// TIA Portal project "TiaPortal_TP_Final_V15.1" (V15.1)

(* hardware
DEVICE "S7-1200 station_1"  S7-1200 Station
   slot 0: "Rack_0"  S7-1200 Rack  Rack  V1.0
   slot 1: "PLC_1"  CPU 1214C AC/DC/Rly  6ES7 214-1BE30-0XB0  V2.0
   slot 3: "AQ 1x12BIT_1"  AQ1 signal board  6ES7 232-4HA30-0XB0  V1.0
*)

// ===== PLC "PLC_1"  CPU 1214C AC/DC/Rly =====

VAR_GLOBAL   // PLC tag table "Tabla de variables estándar"
   "Encendido" AT %M1.4 : Bool;
   "salida_duty_cycle" AT %QW80 : Int;
   "aceleracion_carrito" AT %MD58 : Real;
   "VEL1" AT %I0.2 : Bool;
   "VEL2" AT %I0.3 : Bool;
   "VEL3" AT %I0.4 : Bool;
   "VEL4" AT %I0.5 : Bool;
END_VAR

VAR_GLOBAL   // PLC tag table "Tabla de variables estándar_1"
   "System_Byte" AT %MB1 : Byte;
   "FirstScan" AT %M1.0 : Bool;
   "DiagStatusUpdate" AT %M1.1 : Bool;
   "AlwaysTRUE" AT %M1.2 : Bool;
   "AlwaysFALSE" AT %M1.3 : Bool;
   "Clock_Byte" AT %MB0 : Byte;
   "Clock_10Hz" AT %M0.0 : Bool;
   "Clock_5Hz" AT %M0.1 : Bool;
   "Clock_2.5Hz" AT %M0.2 : Bool;
   "Clock_2Hz" AT %M0.3 : Bool;
   "Clock_1.25Hz" AT %M0.4 : Bool;
   "Clock_1Hz" AT %M0.5 : Bool;
   "Clock_0.625Hz" AT %M0.6 : Bool;
   "Clock_0.5Hz" AT %M0.7 : Bool;
   "tcon_done_save" AT %M2.0 : Bool;
   "lectura_potenciometro" AT %IW66 : Word;
   "lectura_tacometro" AT %IW64 : Word;
   "PM" AT %I0.0 : Bool;
   "PP" AT %I0.1 : Bool;
   "lim_carreraA" AT %I1.3 : Bool;
   "lim_carreraB" AT %I1.2 : Bool;
   "posicion_carrito" AT %MD50 : Real;
   "velocidad_carrito" AT %MD54 : Real;
END_VAR

VAR_GLOBAL CONSTANT   // PLC tag table "Tabla de variables estándar_1"
   "Ninguno" : Pip := 65535;
   "Actualización automática" : Pip := 0;
   "IPP 1" : Pip := 1;
   "IPP 2" : Pip := 2;
   "IPP 3" : Pip := 3;
   "IPP 4" : Pip := 4;
   "IPP OB Servo" : Pip := 32768;
   "Local~MC" : Hw_SubModule := 51;
   "Local~Common" : Hw_SubModule := 50;
   "Local~Device" : Hw_Device := 32;
   "Local~Configuration" : Hw_SubModule := 33;
   "Local~Exec" : Hw_SubModule := 52;
   "Local(1)" : Hw_SubModule := 49;
   "Local~Interfaz_PROFINET_1(1)" : Hw_Interface := 64;
   "Local~Interfaz_PROFINET_1~Puerto_1(1)" : Hw_Interface := 65;
   "Local~Interfaz_PROFINET_1~Puerto_2" : Hw_Interface := 66;
   "Local~HSC_1(1)" : Hw_Hsc := 257;
   "Local~HSC_2(1)" : Hw_Hsc := 258;
   "Local~HSC_3(1)" : Hw_Hsc := 259;
   "Local~HSC_4(1)" : Hw_Hsc := 260;
   "Local~HSC_5(1)" : Hw_Hsc := 261;
   "Local~HSC_6(1)" : Hw_Hsc := 262;
   "Local~AI_2_AQ_2_1" : Hw_SubModule := 263;
   "Local~DI_14_DQ_10_1(1)" : Hw_SubModule := 264;
   "Local~Pulse_1(1)" : Hw_Pwm := 265;
   "Local~Pulse_2(1)" : Hw_Pwm := 266;
   "Local~Pulse_3" : Hw_Pwm := 267;
   "Local~Pulse_4" : Hw_Pwm := 268;
   "OB_Main(1)" : OB_PCYCLE := 1;
END_VAR

DATA_BLOCK "Datos_TSEND"   // DB2
{ S7_Optimized_Access := 'TRUE' }
VERSION : 0.1
   VAR
      data : Struct
         u : Real;
         aceleracion_carrito : Real;
         duty_cycle_pwm : Int;
      END_STRUCT;
   END_VAR
BEGIN
END_DATA_BLOCK

DATA_BLOCK "Comunicacion_DB"   // DB7
{ S7_Optimized_Access := 'TRUE' }
VERSION : 0.1
// stored: InstanceOfName Comunicacion
"Comunicacion"
BEGIN
END_DATA_BLOCK

DATA_BLOCK "Integrador_Velocidad_DB"   // DB9
{ S7_Optimized_Access := 'TRUE' }
VERSION : 0.1
// stored: InstanceOfName Integrador
"Integrador"
BEGIN
END_DATA_BLOCK

DATA_BLOCK "Controlador_DB"   // DB10
{ S7_Optimized_Access := 'TRUE' }
VERSION : 0.1
// stored: InstanceOfName Controlador
"Controlador"
BEGIN
END_DATA_BLOCK

DATA_BLOCK "Datos_General"   // DB11
{ S7_Optimized_Access := 'TRUE' }
VERSION : 0.1
   VAR
      MIN_ACEL_CARRITO : Real := -100.0;   // Aceleración mínima del carrito (porcentaje)
      MAX_ACEL_CARRITO : Real := 100.0;   // Aceleración máxima del carrito (porcentaje)
      MIN_VEL_CARRITO : Real := -100.0;   // Velocidad minima de motor (porcentaje)
      MAX_VEL_CARRITO : Real := 100.0;   // Velocidad maxima del carrito (porcentaje)
      MIN_POS_CARRITO : Real := -160.0;   // Posicion minima del carrito (en mm)
      MAX_POS_CARRITO : Real := 160.0;   // Posicion maxima del carrito (en mm)
      INIT_VEL_RESET : Real := 0.0;   // Velocidad inicial al resetear (porcentaje)
      INIT_POS_RESET : Real := 0.0;   // Posicion inicial al resetear (en mm)
      Tiempo_Muestreo : Real := 0.01;   // Tiempo en segundos del OB30
      LIM_INF_FILTRO_ACEL : Real := -5.0;   // Límite inferior del filtro para la aceleración
      LIM_SUP_FILTRO_ACEL : Real := 5.0;   // Límite superior del filtro para la aceleración
      SP_VEL_CARRITO : Real := 30.0;   // Set Point de velocidad del carrito
   END_VAR
BEGIN
END_DATA_BLOCK

DATA_BLOCK "Rutina_Identificacion_DB"   // DB12
{ S7_Optimized_Access := 'TRUE' }
VERSION : 0.1
// stored: InstanceOfName Rutina_Identificacion
"Rutina_Identificacion"
BEGIN
END_DATA_BLOCK

// folder: System blocks/Program resources

DATA_BLOCK "PLC_CONECTION_DB_"   // DB6
{ S7_Optimized_Access := 'TRUE' }
AUTHOR : SIMATIC
FAMILY : MC7Plus
NAME : TCON_Prm
VERSION : 1.0
// stored: InstanceOfName TCON_Param
"TCON_Param"
BEGIN
   ID := 2;
   REM_TSAP_ID[1] := B#16#07;
   REM_TSAP_ID[2] := B#16#D0;
   REM_STADDR[1] := 192;
   REM_STADDR[2] := 168;
   REM_STADDR[3] := 2;
   REM_STADDR[4] := 241;
END_DATA_BLOCK

// folder: (top level)

FUNCTION_BLOCK "Comunicacion"   // FB1, LAD
{ S7_Optimized_Access := 'TRUE' }
VERSION : 0.1
   VAR_INPUT
      acel_carrito : Real;
      vel_carrito : Real;
      salida_pwm : Int;
      vel_comandada : Real;
   END_VAR
   VAR CONSTANT
      LEN_DATA : UInt := 10;
   END_VAR
BEGIN

REGION Network 1
   // Se busca la conexión con la PC 1 vez por segundo
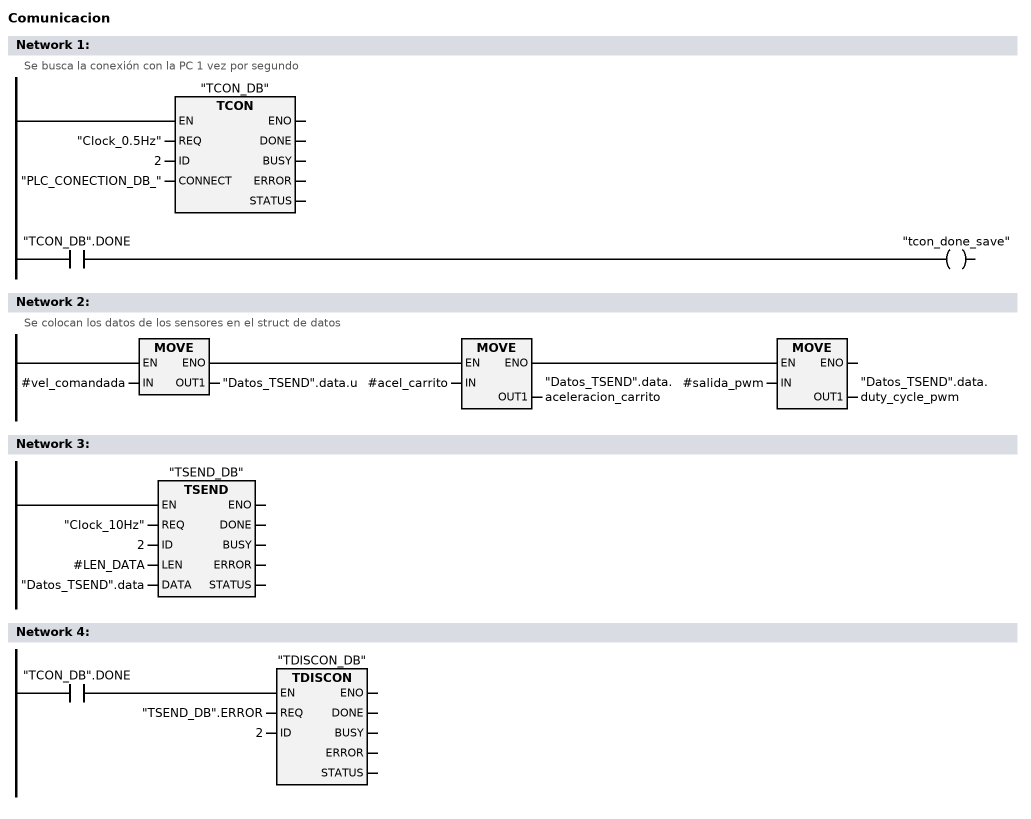
   "TCON_DB"(REQ := "Clock_0.5Hz", ID := 2, CONNECT := "PLC_CONECTION_DB_");   // TCON
   "tcon_done_save" := "TCON_DB".DONE;
END_REGION

REGION Network 2
   // Se colocan los datos de los sensores en el struct de datos
   RUNG wire#powerrail
      { S7_GenerateENO := "TRUE" } Move(in := #vel_comandada, out1 => "Datos_TSEND".data.u)
      { S7_GenerateENO := "TRUE" } Move(in := #acel_carrito, out1 => "Datos_TSEND".data.aceleracion_carrito)
      { S7_GenerateENO := "TRUE" } Move(in := #salida_pwm, out1 => "Datos_TSEND".data.duty_cycle_pwm)
   END_RUNG
   // the same network as SCL:
   // ENO of a box is taken as its EN; it also drops when the box reports an error
   "Datos_TSEND".data.u := #vel_comandada;
   "Datos_TSEND".data.aceleracion_carrito := #acel_carrito;
   "Datos_TSEND".data.duty_cycle_pwm := #salida_pwm;
END_REGION

REGION Network 3
   "TSEND_DB"(REQ := "Clock_10Hz", ID := 2, LEN := #LEN_DATA, DATA := "Datos_TSEND".data);   // TSEND
END_REGION

REGION Network 4
   IF "TCON_DB".DONE THEN
       "TDISCON_DB"(REQ := "TSEND_DB".ERROR, ID := 2);   // TDISCON
   END_IF;
END_REGION
END_FUNCTION_BLOCK

FUNCTION_BLOCK "Controlador"   // FB2, LAD
{ S7_Optimized_Access := 'TRUE' }
VERSION : 0.1
   VAR_INPUT
      SP_Velocidad : Real;   // en mm
      velocidad_actual_carrito : Real;   // porcentaje
      min_vel_perc_carrito : Real;   // porcentaje
      max_vel_perc_carrito : Real;   // porcentaje
   END_VAR
   VAR_OUTPUT
      salida_motor : Int;   // un valor entre n_cuenta_min y n_cuenta_max
   END_VAR
   VAR_TEMP
      vel_carrito_perc_pid : Real;
      vel : Real;
      vel_carrito_norm_pid : Real;
   END_VAR
   VAR CONSTANT
      n_cuenta_min : Int := 0;
      n_cuenta_max : Int := 27648;   // correspondiente a 16 bits del mapeo
   END_VAR
BEGIN

REGION Network 1
   // PID_VELOCIDAD
   // 
   // Input:
   // Recibe la velocidad actual del carrito en porcentaje y el setpoint en porcentaje (ambos son reales de -100.0 a 100.0)
   // 
   // Output:
   // Genera una salida porcentual entre -100.0%  y 100.0%, que es la velocidad a la cual debe accionarse el motor en reversa o en directa respectivamente.
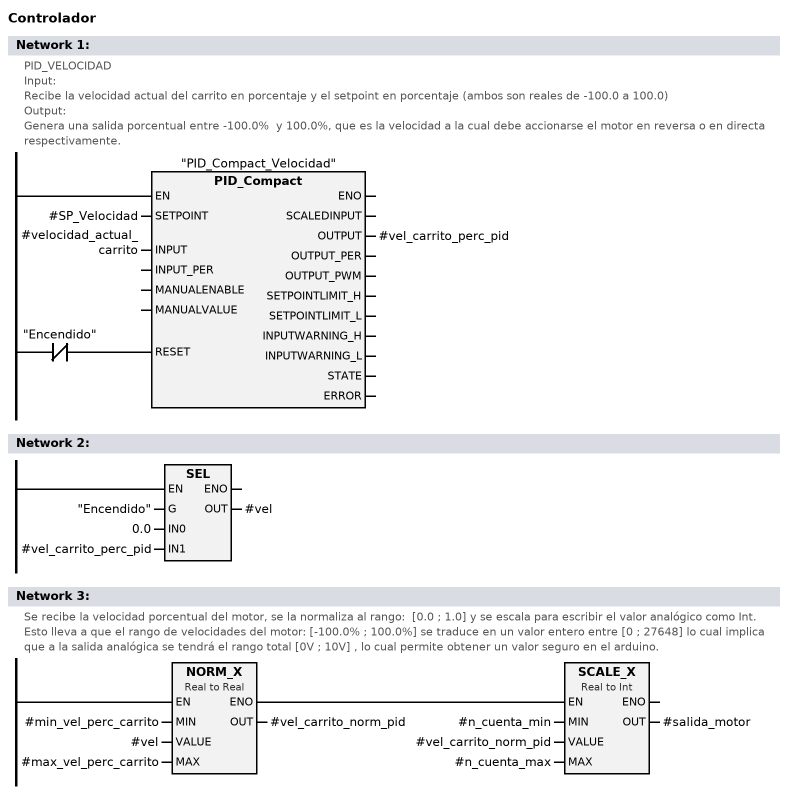
   "PID_Compact_Velocidad"(Setpoint := #SP_Velocidad,   // PID_Compact
                           Input := #velocidad_actual_carrito,
                           Reset := NOT "Encendido",
                           Output => #vel_carrito_perc_pid);
END_REGION

REGION Network 2
   #vel := SEL(G := "Encendido", IN0 := 0.0, IN1 := #vel_carrito_perc_pid);
END_REGION

REGION Network 3
   // Se recibe la velocidad porcentual del motor, se la normaliza al rango:  [0.0 ; 1.0] y se escala para escribir el valor analógico como Int.
   // Esto lleva a que el rango de velocidades del motor: [-100.0% ; 100.0%] se traduce en un valor entero entre [0 ; 27648] lo cual implica que a la salida analógica se tendrá el rango total [0V ; 10V] , lo cual permite obtener un valor seguro en el arduino.
   RUNG wire#powerrail
      { S7_Templates := "[SrcType := Real, DestType := Real]"; S7_GenerateENO := "TRUE" } Normalize(min := #min_vel_perc_carrito, value := #vel, max := #max_vel_perc_carrito, out => #vel_carrito_norm_pid)
      { S7_Templates := "[SrcType := Real, DestType := Int]"; S7_GenerateENO := "TRUE" } Scale(min := #n_cuenta_min, value := #vel_carrito_norm_pid, max := #n_cuenta_max, out => #salida_motor)
   END_RUNG
   // the same network as SCL:
   // ENO of a box is taken as its EN; it also drops when the box reports an error
   #vel_carrito_norm_pid := NORM_X(MIN := #min_vel_perc_carrito, VALUE := #vel, MAX := #max_vel_perc_carrito);
   #salida_motor := SCALE_X(MIN := #n_cuenta_min, VALUE := #vel_carrito_norm_pid, MAX := #n_cuenta_max);
END_REGION
END_FUNCTION_BLOCK

FUNCTION_BLOCK "Rutina_Identificacion"   // FB3, LAD
{ S7_Optimized_Access := 'TRUE' }
VERSION : 0.1
// Se fijó una tolerancia de 20mm para cada movimiento, además de un reinicio automático de la rutina
   VAR_INPUT
      posicion_carrito : Real;
      Encendido : Bool;
   END_VAR
   VAR_OUTPUT
      dc_pwm : Int := 13824;   // (detenido)
   END_VAR
   VAR
      Paso_1 : Bool;
      Paso_2 : Bool;
      Paso_3 : Bool;
      Paso_4 : Bool;
      Paso_5 : Bool;
      Paso_6 : Bool;
      Paso_7 : Bool;
      Paso_8 : Bool;
      Paso_9 : Bool;
      Paso_10 : Bool;
      Paso_11 : Bool;
      Paso_12 : Bool;
      Apagado : Bool;
      aux_encendido : Bool;
      IEC_Timer_Stop_Instance : TON_TIME;
      dc_stop : Int := 13824;   // (detenido)
      dc_f1 : Int := 20000;
      dc_f2 : Int := 19000;
      dc_f3 : Int := 18000;
      dc_b1 : Int := 6500;
      dc_b2 : Int := 7000;
      dc_b3 : Int := 7500;
      IEC_Timer_rutina : TON_TIME;
   END_VAR
   VAR_TEMP   // added for the SCL form of the ladder/FBD networks
      _w1 : Bool;
   END_VAR
   // IEC_Timer_Stop_Instance.PT := T#500ms;
   // IEC_Timer_rutina.PT := T#200ms;
BEGIN

REGION Network 1
   // Inicialización
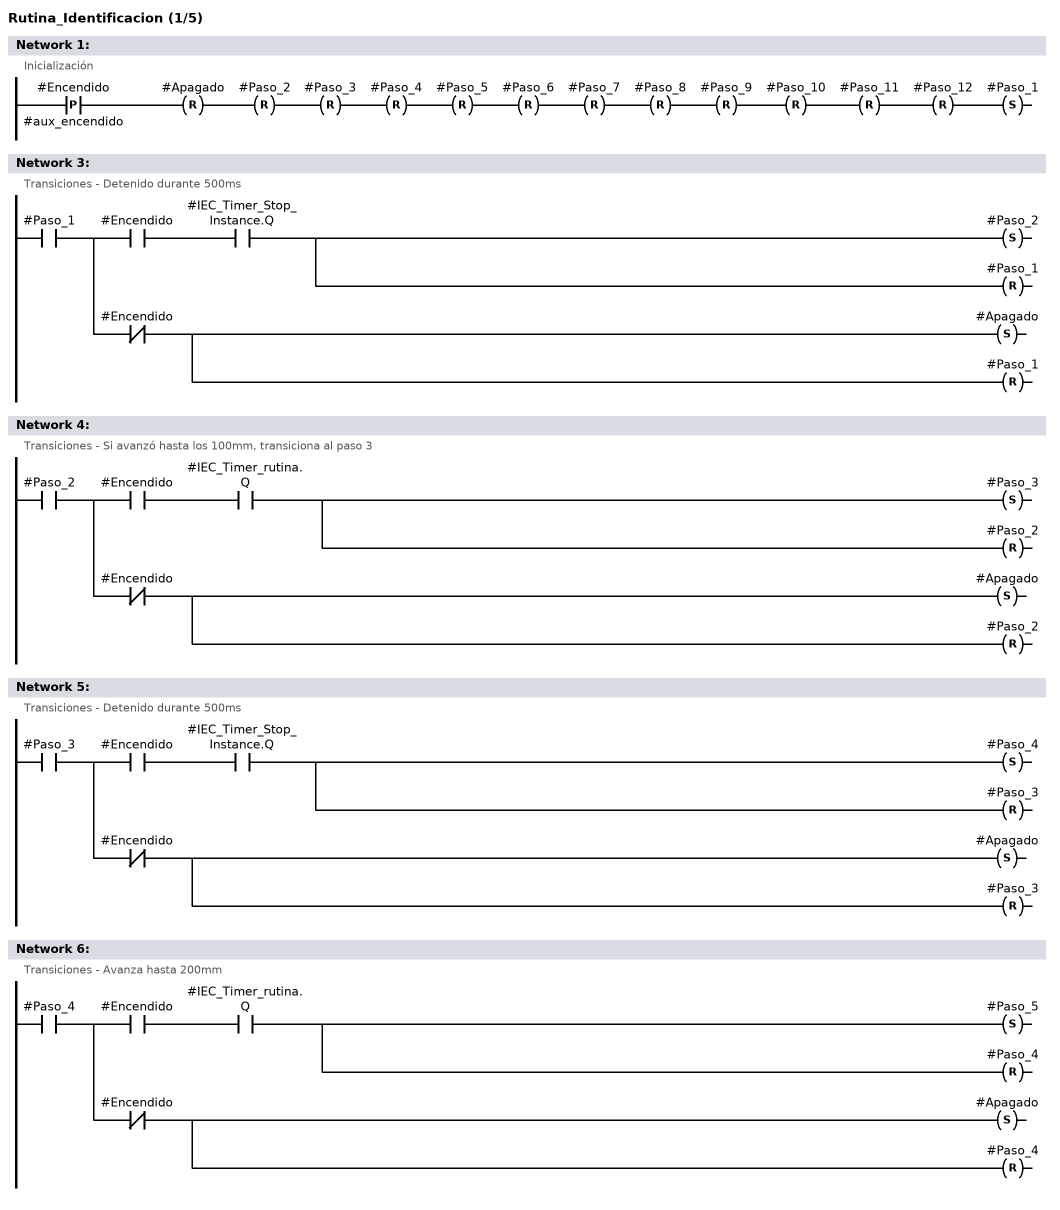
   RUNG wire#powerrail
      P_Contact(operand := #Encendido, bit := #aux_encendido)
      R_Coil( #Apagado )
      R_Coil( #Paso_2 )
      R_Coil( #Paso_3 )
      R_Coil( #Paso_4 )
      R_Coil( #Paso_5 )
      R_Coil( #Paso_6 )
      R_Coil( #Paso_7 )
      R_Coil( #Paso_8 )
      R_Coil( #Paso_9 )
      R_Coil( #Paso_10 )
      R_Coil( #Paso_11 )
      R_Coil( #Paso_12 )
      S_Coil( #Paso_1 )
   END_RUNG
   // the same network as SCL:
   #_w1 := #Encendido AND NOT #aux_encendido;   // rising edge of #Encendido
   #aux_encendido := #Encendido;
   IF #_w1 THEN
       #Apagado := FALSE;
       #Paso_2 := FALSE;
       #Paso_3 := FALSE;
       #Paso_4 := FALSE;
       #Paso_5 := FALSE;
       #Paso_6 := FALSE;
       #Paso_7 := FALSE;
       #Paso_8 := FALSE;
       #Paso_9 := FALSE;
       #Paso_10 := FALSE;
       #Paso_11 := FALSE;
       #Paso_12 := FALSE;
       #Paso_1 := TRUE;
   END_IF;
END_REGION

REGION Network 3
   // Transiciones - Detenido durante 500ms
   RUNG wire#powerrail
      Contact( #Paso_1 )
      wire#w1
      Contact( #Encendido )
      Contact( #IEC_Timer_Stop_Instance.Q )
      wire#w2
      S_Coil( #Paso_2 )
   END_RUNG
   RUNG wire#w2
      R_Coil( #Paso_1 )
   END_RUNG
   RUNG wire#w1
      I_Contact( #Encendido )
      wire#w3
      S_Coil( #Apagado )
   END_RUNG
   RUNG wire#w3
      R_Coil( #Paso_1 )
   END_RUNG
   // the same network as SCL:
   IF #Paso_1 AND #Encendido AND #IEC_Timer_Stop_Instance.Q THEN #Paso_2 := TRUE; END_IF;
   #_w1 := #Paso_1;
   IF #Paso_1 AND #Encendido AND #IEC_Timer_Stop_Instance.Q THEN #Paso_1 := FALSE; END_IF;
   IF #_w1 AND NOT #Encendido THEN
       #Apagado := TRUE;
       #Paso_1 := FALSE;
   END_IF;
END_REGION

REGION Network 4
   // Transiciones - Si avanzó hasta los 100mm, transiciona al paso 3
   RUNG wire#powerrail
      Contact( #Paso_2 )
      wire#w1
      Contact( #Encendido )
      Contact( #IEC_Timer_rutina.Q )
      wire#w2
      S_Coil( #Paso_3 )
   END_RUNG
   RUNG wire#w2
      R_Coil( #Paso_2 )
   END_RUNG
   RUNG wire#w1
      I_Contact( #Encendido )
      wire#w3
      S_Coil( #Apagado )
   END_RUNG
   RUNG wire#w3
      R_Coil( #Paso_2 )
   END_RUNG
   // the same network as SCL:
   IF #Paso_2 AND #Encendido AND #IEC_Timer_rutina.Q THEN #Paso_3 := TRUE; END_IF;
   #_w1 := #Paso_2;
   IF #Paso_2 AND #Encendido AND #IEC_Timer_rutina.Q THEN #Paso_2 := FALSE; END_IF;
   IF #_w1 AND NOT #Encendido THEN
       #Apagado := TRUE;
       #Paso_2 := FALSE;
   END_IF;
END_REGION

REGION Network 5
   // Transiciones - Detenido durante 500ms
   RUNG wire#powerrail
      Contact( #Paso_3 )
      wire#w1
      Contact( #Encendido )
      Contact( #IEC_Timer_Stop_Instance.Q )
      wire#w2
      S_Coil( #Paso_4 )
   END_RUNG
   RUNG wire#w2
      R_Coil( #Paso_3 )
   END_RUNG
   RUNG wire#w1
      I_Contact( #Encendido )
      wire#w3
      S_Coil( #Apagado )
   END_RUNG
   RUNG wire#w3
      R_Coil( #Paso_3 )
   END_RUNG
   // the same network as SCL:
   IF #Paso_3 AND #Encendido AND #IEC_Timer_Stop_Instance.Q THEN #Paso_4 := TRUE; END_IF;
   #_w1 := #Paso_3;
   IF #Paso_3 AND #Encendido AND #IEC_Timer_Stop_Instance.Q THEN #Paso_3 := FALSE; END_IF;
   IF #_w1 AND NOT #Encendido THEN
       #Apagado := TRUE;
       #Paso_3 := FALSE;
   END_IF;
END_REGION

REGION Network 6
   // Transiciones - Avanza hasta 200mm
   RUNG wire#powerrail
      Contact( #Paso_4 )
      wire#w1
      Contact( #Encendido )
      Contact( #IEC_Timer_rutina.Q )
      wire#w2
      S_Coil( #Paso_5 )
   END_RUNG
   RUNG wire#w2
      R_Coil( #Paso_4 )
   END_RUNG
   RUNG wire#w1
      I_Contact( #Encendido )
      wire#w3
      S_Coil( #Apagado )
   END_RUNG
   RUNG wire#w3
      R_Coil( #Paso_4 )
   END_RUNG
   // the same network as SCL:
   IF #Paso_4 AND #Encendido AND #IEC_Timer_rutina.Q THEN #Paso_5 := TRUE; END_IF;
   #_w1 := #Paso_4;
   IF #Paso_4 AND #Encendido AND #IEC_Timer_rutina.Q THEN #Paso_4 := FALSE; END_IF;
   IF #_w1 AND NOT #Encendido THEN
       #Apagado := TRUE;
       #Paso_4 := FALSE;
   END_IF;
END_REGION

REGION Network 7
   // Transiciones - Detenido durante 500ms
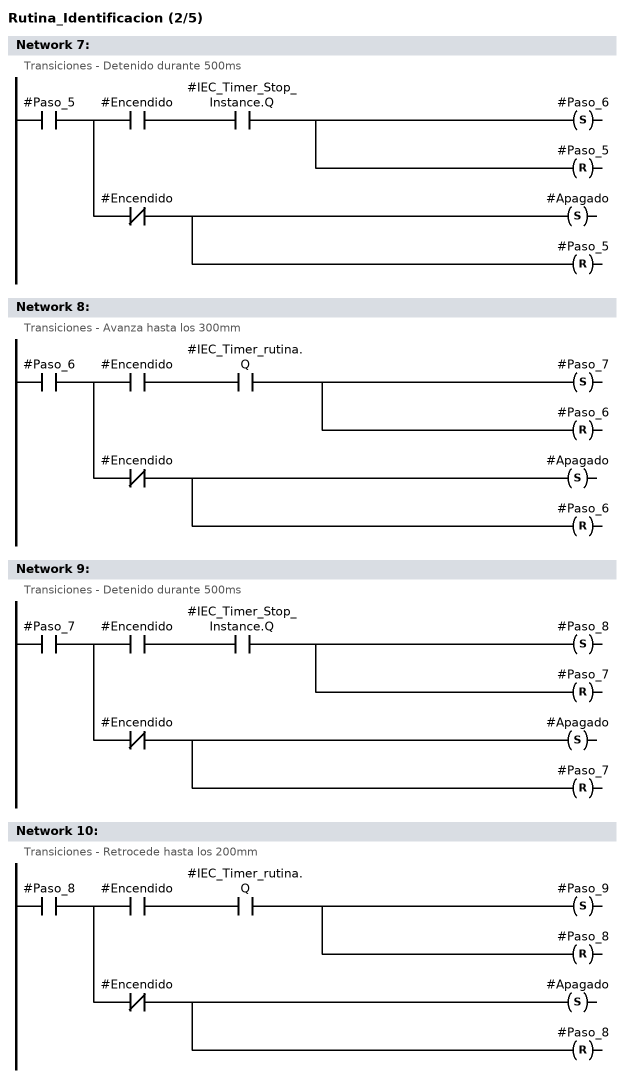
   RUNG wire#powerrail
      Contact( #Paso_5 )
      wire#w1
      Contact( #Encendido )
      Contact( #IEC_Timer_Stop_Instance.Q )
      wire#w2
      S_Coil( #Paso_6 )
   END_RUNG
   RUNG wire#w2
      R_Coil( #Paso_5 )
   END_RUNG
   RUNG wire#w1
      I_Contact( #Encendido )
      wire#w3
      S_Coil( #Apagado )
   END_RUNG
   RUNG wire#w3
      R_Coil( #Paso_5 )
   END_RUNG
   // the same network as SCL:
   IF #Paso_5 AND #Encendido AND #IEC_Timer_Stop_Instance.Q THEN #Paso_6 := TRUE; END_IF;
   #_w1 := #Paso_5;
   IF #Paso_5 AND #Encendido AND #IEC_Timer_Stop_Instance.Q THEN #Paso_5 := FALSE; END_IF;
   IF #_w1 AND NOT #Encendido THEN
       #Apagado := TRUE;
       #Paso_5 := FALSE;
   END_IF;
END_REGION

REGION Network 8
   // Transiciones - Avanza hasta los 300mm
   RUNG wire#powerrail
      Contact( #Paso_6 )
      wire#w1
      Contact( #Encendido )
      Contact( #IEC_Timer_rutina.Q )
      wire#w2
      S_Coil( #Paso_7 )
   END_RUNG
   RUNG wire#w2
      R_Coil( #Paso_6 )
   END_RUNG
   RUNG wire#w1
      I_Contact( #Encendido )
      wire#w3
      S_Coil( #Apagado )
   END_RUNG
   RUNG wire#w3
      R_Coil( #Paso_6 )
   END_RUNG
   // the same network as SCL:
   IF #Paso_6 AND #Encendido AND #IEC_Timer_rutina.Q THEN #Paso_7 := TRUE; END_IF;
   #_w1 := #Paso_6;
   IF #Paso_6 AND #Encendido AND #IEC_Timer_rutina.Q THEN #Paso_6 := FALSE; END_IF;
   IF #_w1 AND NOT #Encendido THEN
       #Apagado := TRUE;
       #Paso_6 := FALSE;
   END_IF;
END_REGION

REGION Network 9
   // Transiciones - Detenido durante 500ms
   RUNG wire#powerrail
      Contact( #Paso_7 )
      wire#w1
      Contact( #Encendido )
      Contact( #IEC_Timer_Stop_Instance.Q )
      wire#w2
      S_Coil( #Paso_8 )
   END_RUNG
   RUNG wire#w2
      R_Coil( #Paso_7 )
   END_RUNG
   RUNG wire#w1
      I_Contact( #Encendido )
      wire#w3
      S_Coil( #Apagado )
   END_RUNG
   RUNG wire#w3
      R_Coil( #Paso_7 )
   END_RUNG
   // the same network as SCL:
   IF #Paso_7 AND #Encendido AND #IEC_Timer_Stop_Instance.Q THEN #Paso_8 := TRUE; END_IF;
   #_w1 := #Paso_7;
   IF #Paso_7 AND #Encendido AND #IEC_Timer_Stop_Instance.Q THEN #Paso_7 := FALSE; END_IF;
   IF #_w1 AND NOT #Encendido THEN
       #Apagado := TRUE;
       #Paso_7 := FALSE;
   END_IF;
END_REGION

REGION Network 10
   // Transiciones - Retrocede hasta los 200mm
   RUNG wire#powerrail
      Contact( #Paso_8 )
      wire#w1
      Contact( #Encendido )
      Contact( #IEC_Timer_rutina.Q )
      wire#w2
      S_Coil( #Paso_9 )
   END_RUNG
   RUNG wire#w2
      R_Coil( #Paso_8 )
   END_RUNG
   RUNG wire#w1
      I_Contact( #Encendido )
      wire#w3
      S_Coil( #Apagado )
   END_RUNG
   RUNG wire#w3
      R_Coil( #Paso_8 )
   END_RUNG
   // the same network as SCL:
   IF #Paso_8 AND #Encendido AND #IEC_Timer_rutina.Q THEN #Paso_9 := TRUE; END_IF;
   #_w1 := #Paso_8;
   IF #Paso_8 AND #Encendido AND #IEC_Timer_rutina.Q THEN #Paso_8 := FALSE; END_IF;
   IF #_w1 AND NOT #Encendido THEN
       #Apagado := TRUE;
       #Paso_8 := FALSE;
   END_IF;
END_REGION

REGION Network 11
   // Transiciones - Detenido durante 500ms
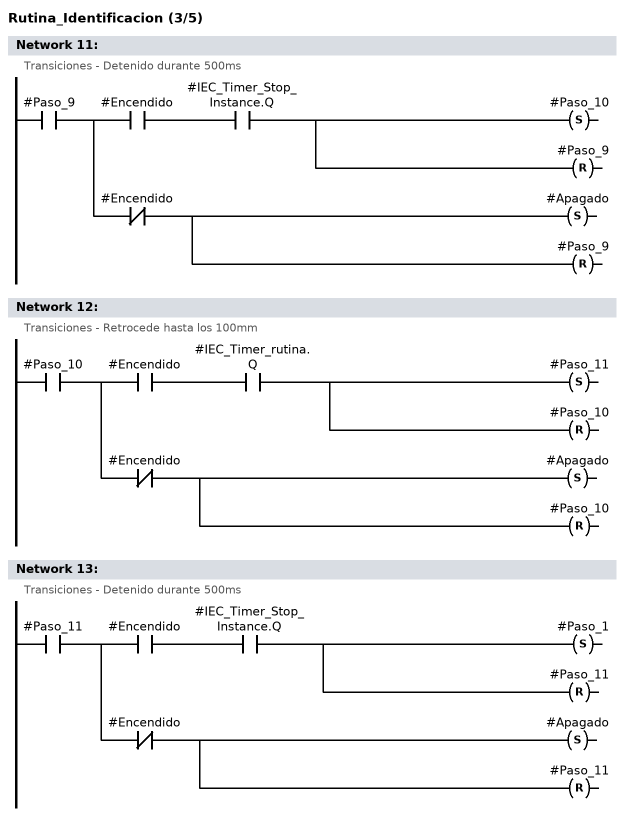
   RUNG wire#powerrail
      Contact( #Paso_9 )
      wire#w1
      Contact( #Encendido )
      Contact( #IEC_Timer_Stop_Instance.Q )
      wire#w2
      S_Coil( #Paso_10 )
   END_RUNG
   RUNG wire#w2
      R_Coil( #Paso_9 )
   END_RUNG
   RUNG wire#w1
      I_Contact( #Encendido )
      wire#w3
      S_Coil( #Apagado )
   END_RUNG
   RUNG wire#w3
      R_Coil( #Paso_9 )
   END_RUNG
   // the same network as SCL:
   IF #Paso_9 AND #Encendido AND #IEC_Timer_Stop_Instance.Q THEN #Paso_10 := TRUE; END_IF;
   #_w1 := #Paso_9;
   IF #Paso_9 AND #Encendido AND #IEC_Timer_Stop_Instance.Q THEN #Paso_9 := FALSE; END_IF;
   IF #_w1 AND NOT #Encendido THEN
       #Apagado := TRUE;
       #Paso_9 := FALSE;
   END_IF;
END_REGION

REGION Network 12
   // Transiciones - Retrocede hasta los 100mm
   RUNG wire#powerrail
      Contact( #Paso_10 )
      wire#w1
      Contact( #Encendido )
      Contact( #IEC_Timer_rutina.Q )
      wire#w2
      S_Coil( #Paso_11 )
   END_RUNG
   RUNG wire#w2
      R_Coil( #Paso_10 )
   END_RUNG
   RUNG wire#w1
      I_Contact( #Encendido )
      wire#w3
      S_Coil( #Apagado )
   END_RUNG
   RUNG wire#w3
      R_Coil( #Paso_10 )
   END_RUNG
   // the same network as SCL:
   IF #Paso_10 AND #Encendido AND #IEC_Timer_rutina.Q THEN #Paso_11 := TRUE; END_IF;
   #_w1 := #Paso_10;
   IF #Paso_10 AND #Encendido AND #IEC_Timer_rutina.Q THEN #Paso_10 := FALSE; END_IF;
   IF #_w1 AND NOT #Encendido THEN
       #Apagado := TRUE;
       #Paso_10 := FALSE;
   END_IF;
END_REGION

REGION Network 13
   // Transiciones - Detenido durante 500ms
   RUNG wire#powerrail
      Contact( #Paso_11 )
      wire#w1
      Contact( #Encendido )
      Contact( #IEC_Timer_Stop_Instance.Q )
      wire#w2
      S_Coil( #Paso_1 )
   END_RUNG
   RUNG wire#w2
      R_Coil( #Paso_11 )
   END_RUNG
   RUNG wire#w1
      I_Contact( #Encendido )
      wire#w3
      S_Coil( #Apagado )
   END_RUNG
   RUNG wire#w3
      R_Coil( #Paso_11 )
   END_RUNG
   // the same network as SCL:
   IF #Paso_11 AND #Encendido AND #IEC_Timer_Stop_Instance.Q THEN #Paso_1 := TRUE; END_IF;
   #_w1 := #Paso_11;
   IF #Paso_11 AND #Encendido AND #IEC_Timer_Stop_Instance.Q THEN #Paso_11 := FALSE; END_IF;
   IF #_w1 AND NOT #Encendido THEN
       #Apagado := TRUE;
       #Paso_11 := FALSE;
   END_IF;
END_REGION

REGION Network 14
   // ACCIONES - AVANCES (f) Y RETROCESOS (b)
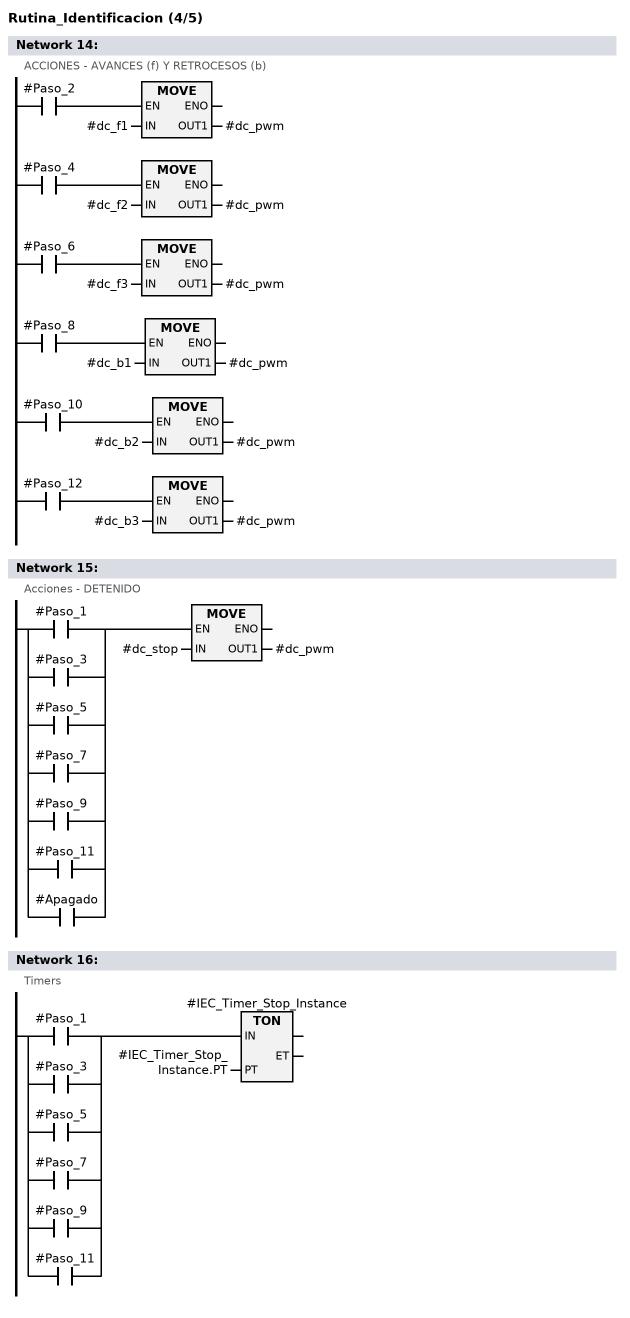
   RUNG wire#powerrail
      Contact( #Paso_2 )
      { S7_GenerateENO := "TRUE" } Move(in := #dc_f1, out1 => #dc_pwm)
   END_RUNG
   RUNG wire#powerrail
      Contact( #Paso_4 )
      { S7_GenerateENO := "TRUE" } Move(in := #dc_f2, out1 => #dc_pwm)
   END_RUNG
   RUNG wire#powerrail
      Contact( #Paso_6 )
      { S7_GenerateENO := "TRUE" } Move(in := #dc_f3, out1 => #dc_pwm)
   END_RUNG
   RUNG wire#powerrail
      Contact( #Paso_8 )
      { S7_GenerateENO := "TRUE" } Move(in := #dc_b1, out1 => #dc_pwm)
   END_RUNG
   RUNG wire#powerrail
      Contact( #Paso_10 )
      { S7_GenerateENO := "TRUE" } Move(in := #dc_b2, out1 => #dc_pwm)
   END_RUNG
   RUNG wire#powerrail
      Contact( #Paso_12 )
      { S7_GenerateENO := "TRUE" } Move(in := #dc_b3, out1 => #dc_pwm)
   END_RUNG
   // the same network as SCL:
   IF #Paso_2 THEN #dc_pwm := #dc_f1; END_IF;
   IF #Paso_4 THEN #dc_pwm := #dc_f2; END_IF;
   IF #Paso_6 THEN #dc_pwm := #dc_f3; END_IF;
   IF #Paso_8 THEN #dc_pwm := #dc_b1; END_IF;
   IF #Paso_10 THEN #dc_pwm := #dc_b2; END_IF;
   IF #Paso_12 THEN #dc_pwm := #dc_b3; END_IF;
END_REGION

REGION Network 15
   // Acciones - DETENIDO
   RUNG wire#powerrail
      Contact( #Paso_1 )
      wire#w1
      { S7_GenerateENO := "TRUE" } Move(in := #dc_stop, out1 => #dc_pwm)
   END_RUNG
   RUNG wire#powerrail
      Contact( #Paso_3 )
   END_RUNG wire#w1
   RUNG wire#powerrail
      Contact( #Paso_5 )
   END_RUNG wire#w1
   RUNG wire#powerrail
      Contact( #Paso_7 )
   END_RUNG wire#w1
   RUNG wire#powerrail
      Contact( #Paso_9 )
   END_RUNG wire#w1
   RUNG wire#powerrail
      Contact( #Paso_11 )
   END_RUNG wire#w1
   RUNG wire#powerrail
      Contact( #Apagado )
   END_RUNG wire#w1
   // the same network as SCL:
   IF #Paso_1 OR #Paso_3 OR #Paso_5 OR #Paso_7 OR #Paso_9 OR #Paso_11 OR #Apagado THEN
       #dc_pwm := #dc_stop;
   END_IF;
END_REGION

REGION Network 16
   // Timers
   #IEC_Timer_Stop_Instance(IN := #Paso_1 OR #Paso_3 OR #Paso_5 OR #Paso_7 OR #Paso_9 OR #Paso_11,   // TON
                           PT := #IEC_Timer_Stop_Instance.PT);
END_REGION

REGION Network 17
   // Timers
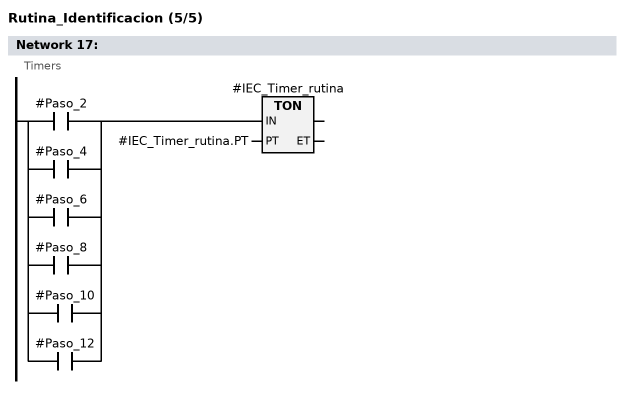
   #IEC_Timer_rutina(IN := #Paso_2 OR #Paso_4 OR #Paso_6 OR #Paso_8 OR #Paso_10 OR #Paso_12,   // TON
                     PT := #IEC_Timer_rutina.PT);
END_REGION
END_FUNCTION_BLOCK

FUNCTION_BLOCK "Integrador"   // FB4, SCL
{ S7_Optimized_Access := 'TRUE' }
VERSION : 0.1
   VAR_INPUT
      in_X : Real;   // señal a integrar
      in_DeltaT : Real;   // periodo de muestreo en seg: 0.01
      in_Reset : Bool;   // para llevar la salida a 0 o su valor inicial
      in_InitValue : Real;   // valor inicial al resetear (0.0 o el valor minimo)
      in_OutMin : Real;   // limite inferior de saturacion
      in_OutMax : Real;   // limite superior de saturacion
      in_Enable : Bool;   // si está en FALSE, congela la salida en el último valor calculado
   END_VAR
   VAR_OUTPUT
      out_Y : Real;   // salida integrada
   END_VAR
   VAR
      stat_Y : Real;   // acumulador interno
      stat_XPrev : Real;   // muestra anterior de la entrada
   END_VAR
BEGIN
   IF #in_Reset THEN
       #stat_Y := #in_InitValue;
       #stat_XPrev := #in_X;
   ELSIF #in_Enable THEN
       // Integracion trapezoidal
       #stat_Y := #stat_Y + ((#in_X + #stat_XPrev) * 0.5) * #in_DeltaT;

       // Limites de saturacion
       IF #stat_Y > #in_OutMax THEN
           #stat_Y := #in_OutMax;
       ELSIF #stat_Y < #in_OutMin THEN
           #stat_Y := #in_OutMin;
       END_IF;

       //Actualización del valor anterior
       #stat_XPrev := #in_X;
   ELSE
       #stat_XPrev := #in_X;
   END_IF;

   #out_Y := #stat_Y;
END_FUNCTION_BLOCK

FUNCTION "a2v" : Void   // FC1, LAD
{ S7_Optimized_Access := 'TRUE' }
VERSION : 0.1
   VAR_INPUT
      "Analog input" : Int;
      K1 : Int;
      K2 : Int;
      Min : Real;
      Max : Real;
   END_VAR
   VAR_OUTPUT
      Value : Real;
   END_VAR
   VAR_TEMP
      "Valor normalizado" : Real;
   END_VAR
BEGIN

REGION Network 1
   // Recibe el rango de datos en el que se encuentra la Entrada a normalizar y el rango de datos en el que se encuentra la variable convertida
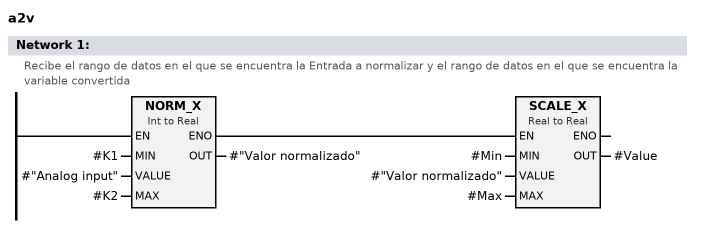
   RUNG wire#powerrail
      { S7_Templates := "[SrcType := Int, DestType := Real]"; S7_GenerateENO := "TRUE" } Normalize(min := #K1, value := #"Analog input", max := #K2, out => #"Valor normalizado")
      { S7_Templates := "[SrcType := Real, DestType := Real]"; S7_GenerateENO := "TRUE" } Scale(min := #Min, value := #"Valor normalizado", max := #Max, out => #Value)
   END_RUNG
   // the same network as SCL:
   // ENO of a box is taken as its EN; it also drops when the box reports an error
   #"Valor normalizado" := NORM_X(MIN := #K1, VALUE := #"Analog input", MAX := #K2);
   #Value := SCALE_X(MIN := #Min, VALUE := #"Valor normalizado", MAX := #Max);
END_REGION
END_FUNCTION

ORGANIZATION_BLOCK "Main"   // OB1, LAD, ProgramCycle
TITLE = "Main Program Sweep (Cycle)"
{ S7_Optimized_Access := 'TRUE' }
VERSION : 0.1
BEGIN

REGION Network 1
   // Marcha / Parada
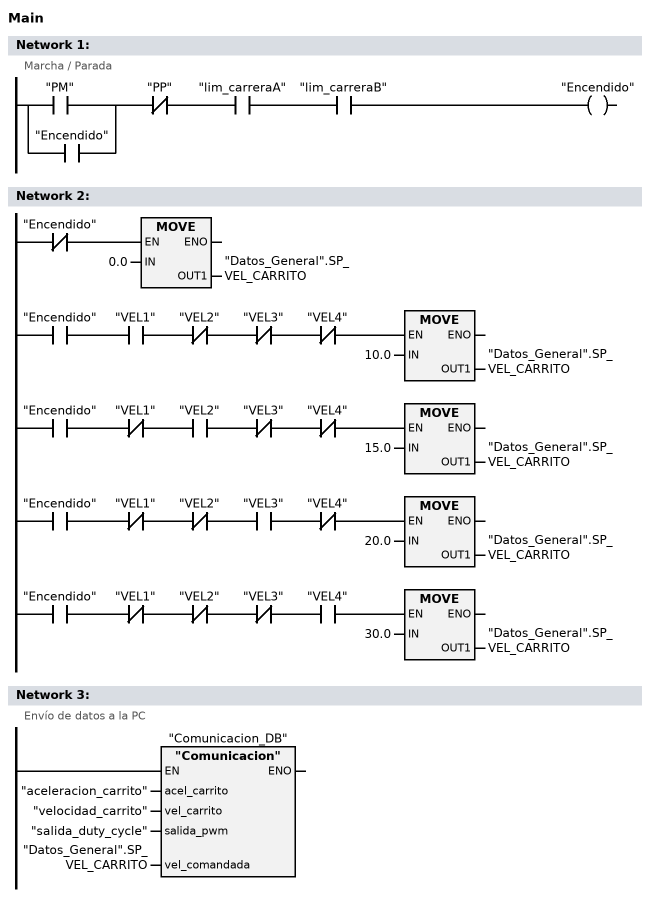
   RUNG wire#powerrail
      Contact( "PM" )
      wire#w1
      I_Contact( "PP" )
      Contact( "lim_carreraA" )
      Contact( "lim_carreraB" )
      Coil( "Encendido" )
   END_RUNG
   RUNG wire#powerrail
      Contact( "Encendido" )
   END_RUNG wire#w1
   // the same network as SCL:
   "Encendido" := ("PM" OR "Encendido") AND NOT "PP" AND "lim_carreraA" AND "lim_carreraB";
END_REGION

REGION Network 2
   RUNG wire#powerrail
      I_Contact( "Encendido" )
      { S7_GenerateENO := "TRUE" } Move(in := 0.0, out1 => "Datos_General".SP_VEL_CARRITO)
   END_RUNG
   RUNG wire#powerrail
      Contact( "Encendido" )
      Contact( "VEL1" )
      I_Contact( "VEL2" )
      I_Contact( "VEL3" )
      I_Contact( "VEL4" )
      { S7_GenerateENO := "TRUE" } Move(in := 10.0, out1 => "Datos_General".SP_VEL_CARRITO)
   END_RUNG
   RUNG wire#powerrail
      Contact( "Encendido" )
      I_Contact( "VEL1" )
      Contact( "VEL2" )
      I_Contact( "VEL3" )
      I_Contact( "VEL4" )
      { S7_GenerateENO := "TRUE" } Move(in := 15.0, out1 => "Datos_General".SP_VEL_CARRITO)
   END_RUNG
   RUNG wire#powerrail
      Contact( "Encendido" )
      I_Contact( "VEL1" )
      I_Contact( "VEL2" )
      Contact( "VEL3" )
      I_Contact( "VEL4" )
      { S7_GenerateENO := "TRUE" } Move(in := 20.0, out1 => "Datos_General".SP_VEL_CARRITO)
   END_RUNG
   RUNG wire#powerrail
      Contact( "Encendido" )
      I_Contact( "VEL1" )
      I_Contact( "VEL2" )
      I_Contact( "VEL3" )
      Contact( "VEL4" )
      { S7_GenerateENO := "TRUE" } Move(in := 30.0, out1 => "Datos_General".SP_VEL_CARRITO)
   END_RUNG
   // the same network as SCL:
   IF NOT "Encendido" THEN "Datos_General".SP_VEL_CARRITO := 0.0; END_IF;
   IF "Encendido" AND "VEL1" AND NOT "VEL2" AND NOT "VEL3" AND NOT "VEL4" THEN
       "Datos_General".SP_VEL_CARRITO := 10.0;
   END_IF;
   IF "Encendido" AND NOT "VEL1" AND "VEL2" AND NOT "VEL3" AND NOT "VEL4" THEN
       "Datos_General".SP_VEL_CARRITO := 15.0;
   END_IF;
   IF "Encendido" AND NOT "VEL1" AND NOT "VEL2" AND "VEL3" AND NOT "VEL4" THEN
       "Datos_General".SP_VEL_CARRITO := 20.0;
   END_IF;
   IF "Encendido" AND NOT "VEL1" AND NOT "VEL2" AND NOT "VEL3" AND "VEL4" THEN
       "Datos_General".SP_VEL_CARRITO := 30.0;
   END_IF;
END_REGION

REGION Network 3
   // Envío de datos a la PC
   RUNG wire#powerrail
      "Comunicacion_DB"(acel_carrito := "aceleracion_carrito", vel_carrito := "velocidad_carrito", salida_pwm := "salida_duty_cycle", vel_comandada := "Datos_General".SP_VEL_CARRITO)
   END_RUNG
   // the same network as SCL:
   "Comunicacion_DB"(acel_carrito := "aceleracion_carrito",   // "Comunicacion"
                     vel_carrito := "velocidad_carrito",
                     salida_pwm := "salida_duty_cycle",
                     vel_comandada := "Datos_General".SP_VEL_CARRITO);
END_REGION
END_ORGANIZATION_BLOCK

ORGANIZATION_BLOCK "Lazo_Control"   // OB30, LAD, CyclicInterrupt
{ S7_Optimized_Access := 'TRUE' }
VERSION : 0.1
   VAR_TEMP
      aceleracion_carrito_sin_filtrar : Real;   // dato de la aceleración convertido, sin filtrar
      SP : Real;
   END_VAR
   VAR CONSTANT
      n_cuenta_min : Int := 0;
      n_cuenta_max : Int := 27648;   // Entrada analógica de 10bits
   END_VAR
BEGIN

REGION Network 1
   // Conversión de la posición del carrito obtenida a partir del sensor
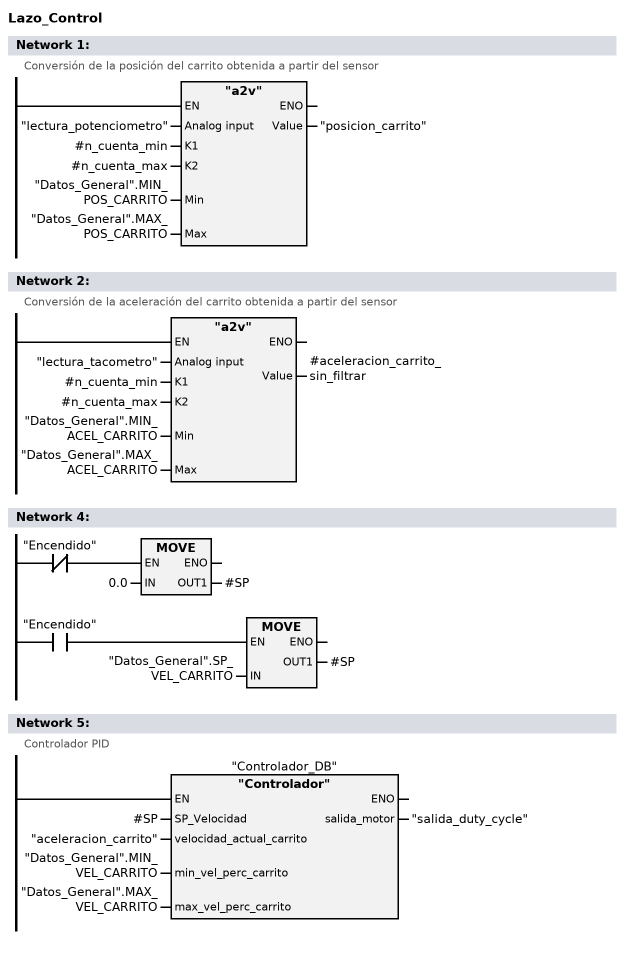
   RUNG wire#powerrail
      "a2v"("Analog input" := "lectura_potenciometro", K1 := #n_cuenta_min, K2 := #n_cuenta_max, Min := "Datos_General".MIN_POS_CARRITO, Max := "Datos_General".MAX_POS_CARRITO, Value => "posicion_carrito")
   END_RUNG
   // the same network as SCL:
   "a2v"("Analog input" := "lectura_potenciometro",
         K1 := #n_cuenta_min,
         K2 := #n_cuenta_max,
         Min := "Datos_General".MIN_POS_CARRITO,
         Max := "Datos_General".MAX_POS_CARRITO,
         Value => "posicion_carrito");
END_REGION

REGION Network 2
   // Conversión de la aceleración del carrito obtenida a partir del sensor
   RUNG wire#powerrail
      "a2v"("Analog input" := "lectura_tacometro", K1 := #n_cuenta_min, K2 := #n_cuenta_max, Min := "Datos_General".MIN_ACEL_CARRITO, Max := "Datos_General".MAX_ACEL_CARRITO, Value => #aceleracion_carrito_sin_filtrar)
   END_RUNG
   // the same network as SCL:
   "a2v"("Analog input" := "lectura_tacometro",
         K1 := #n_cuenta_min,
         K2 := #n_cuenta_max,
         Min := "Datos_General".MIN_ACEL_CARRITO,
         Max := "Datos_General".MAX_ACEL_CARRITO,
         Value => #aceleracion_carrito_sin_filtrar);
END_REGION

REGION Network 3 (SCL): dato de la aceleración convertido, sin filtrar
   // Filtrado de la aceleración del carrito para establecer una zona muerta
   IF (#aceleracion_carrito_sin_filtrar <= "Datos_General".LIM_INF_FILTRO_ACEL) OR (#aceleracion_carrito_sin_filtrar >= "Datos_General".LIM_SUP_FILTRO_ACEL) THEN
       "aceleracion_carrito" := #aceleracion_carrito_sin_filtrar;
   ELSE
       "aceleracion_carrito" := 0.0;
   END_IF;
END_REGION

REGION Network 4
   RUNG wire#powerrail
      I_Contact( "Encendido" )
      { S7_GenerateENO := "TRUE" } Move(in := 0.0, out1 => #SP)
   END_RUNG
   RUNG wire#powerrail
      Contact( "Encendido" )
      { S7_GenerateENO := "TRUE" } Move(in := "Datos_General".SP_VEL_CARRITO, out1 => #SP)
   END_RUNG
   // the same network as SCL:
   IF NOT "Encendido" THEN #SP := 0.0; END_IF;
   IF "Encendido" THEN #SP := "Datos_General".SP_VEL_CARRITO; END_IF;
END_REGION

REGION Network 5
   // Controlador PID
   RUNG wire#powerrail
      "Controlador_DB"(SP_Velocidad := #SP, velocidad_actual_carrito := "aceleracion_carrito", min_vel_perc_carrito := "Datos_General".MIN_VEL_CARRITO, max_vel_perc_carrito := "Datos_General".MAX_VEL_CARRITO, salida_motor => "salida_duty_cycle")
   END_RUNG
   // the same network as SCL:
   "Controlador_DB"(SP_Velocidad := #SP,   // "Controlador"
                    velocidad_actual_carrito := "aceleracion_carrito",
                    min_vel_perc_carrito := "Datos_General".MIN_VEL_CARRITO,
                    max_vel_perc_carrito := "Datos_General".MAX_VEL_CARRITO,
                    salida_motor => "salida_duty_cycle");
END_REGION
END_ORGANIZATION_BLOCK